// TIA Portal V19 export
TYPE "C106_VAR_IF_REL_TYPIC"
   STRUCT
      ALM { ExternalAccessible := 'False'; ExternalVisible := 'False'; ExternalWritable := 'False'} : Bool;   // Alarm per beveiligingsrelais per uitschakelbevel: TRUE = OK / FALSE = Alarm
      AUT_TOE { ExternalAccessible := 'False'; ExternalVisible := 'False'; ExternalWritable := 'False'} : Bool;   // Vermogenschakelaar TOE (gesloten)
      SCA_TOE { ExternalAccessible := 'False'; ExternalVisible := 'False'; ExternalWritable := 'False'} : Bool;   // Aardingschakelaar TOE (gesloten)
      SYNC { ExternalAccessible := 'False'; ExternalVisible := 'False'; ExternalWritable := 'False'} : Bool;   // Lijndifferentieel beveiligingsrelais loopt synchroon
      EXT_AUT { ExternalAccessible := 'False'; ExternalVisible := 'False'; ExternalWritable := 'False'} : Bool;   // Externe (hoofd) beveiliging aangesproken
      EXT_HW { ExternalAccessible := 'False'; ExternalVisible := 'False'; ExternalWritable := 'False'} : Bool;   // Sturings hardware (PLC) in storing
   END_STRUCT;
END_TYPE
